KUKA KRL program: p01.src, p01.dat

--- p01.src ---
&ACCESS RV1
&REL 82
&COMMENT CX482 FHEV
&PARAM EDITMASK = *
&PARAM TEMPLATE = C:\KRC\Roboter\Template\vorgabe
&PARAM DISKPATH = KRC:\R1\Program\Main Programs
DEF p01( )
;================================================
;FOLD INI;%{PE}
  ;FOLD BASISTECH INI
    GLOBAL INTERRUPT DECL 3 WHEN $STOPMESS==TRUE DO IR_STOPM ( )
    INTERRUPT ON 3
    BAS (#INITMOV,0 )
  ;ENDFOLD (BASISTECH INI)
  ;FOLD USER INI
    ;Make your modifications here
BACKJUMP=FALSE
  ;ENDFOLD (USER INI)
;ENDFOLD (INI)
; MODEL     : CX482
; IE GROUP  : FHEV
; STATION   : ST105
; ROBOT     : 105R1
; FUNCTION  : GLUE ON FLANGE - 2C
;================================================

;Control TC
$TIMER[7]=0
$TIMER_STOP[7]=FALSE

;FOLD PTP HOME Vel=100 % DEFAULT;%{PE}%R 8.3.48,%MKUKATPBASIS,%CMOVE,%VPTP,%P 1:PTP, 2:HOME, 3:, 5:100, 7:DEFAULT
$BWDSTART=FALSE
PDAT_ACT=PDEFAULT
FDAT_ACT=FHOME
BAS(#PTP_PARAMS,100)
$H_POS=XHOME
PTP XHOME
;ENDFOLD

;FOLD Start Cycle Timer
$TIMER[1]=0
$TIMER_STOP[1]=FALSE
;ENDFOLD

INFOPOS:
;FOLD PTP P1wait Vel=100 % PDAT2 Tool[5] Base[0];%{PE}%R 8.3.48,%MKUKATPBASIS,%CMOVE,%VPTP,%P 1:PTP, 2:P1wait, 3:, 5:100, 7:PDAT2
$BWDSTART=FALSE
PDAT_ACT=PPDAT2
FDAT_ACT=FP1wait
BAS(#PTP_PARAMS,100)
PTP XP1wait
;ENDFOLD

;if false then

;FOLD TYPE INFO

O_TYPE_REQ=FALSE
WAIT FOR I_TYPE_INFO==0
O_TYPE_REQ=TRUE
WAIT FOR (I_TYPE_INFO>0)
O_TYPE_INFO=I_TYPE_INFO


;ENDFOLD

;rack1 o rack2

;endif

WAIT FOR ($IN[49]==TRUE) OR ($IN[50]==TRUE) OR ($IN[51]==TRUE)

cils_init()
IF $in[49]==TRUE THEN
   INDICE_RACK=1              ;Variable calculo TC
   P01pick1 ( )               ; PICK In Station XX
   IF I_Rethp THEN              ; Return To Home
     GOTO HOMEPOS
   ENDIF
   IF BACKJUMP THEN
     BACKJUMP=FALSE
     GOTO INFOPOS
   ENDIF
   IF CARTJUMP THEN              ; Return To Home
     GOTO HOMEPOS
   ENDIF

  ; P01drop()
   P01drop_new()

endif

IF $in[50]==TRUE THEN
   INDICE_RACK=2              ;Variable calculo TC
   P01pick2 ( )                ; PICK In Station XX
   IF I_Rethp THEN              ; Return To Home
     GOTO HOMEPOS
   ENDIF
   IF BACKJUMP THEN
     BACKJUMP=FALSE
     GOTO INFOPOS
   ENDIF
   IF CARTJUMP THEN              ; Return To Home
     GOTO HOMEPOS
   ENDIF
  ; P01drop()
   P01drop_new()

ENDIF


IF $in[51]==TRUE THEN

   P01pick3 ( )                ; PICK In carton XX


;FOLD OUT 21 'Area Release 5' State=TRUE ;%{PE}%R 8.3.48,%MKUKATPBASIS,%COUT,%VOUTX,%P 2:21, 3:Area Release 5, 5:TRUE, 6:
$OUT[21]=TRUE
;ENDFOLD
;FOLD TYPE INFO

O_TYPE_REQ=FALSE
WAIT FOR I_TYPE_INFO==0
O_TYPE_REQ=TRUE
WAIT FOR (I_TYPE_INFO>0)
POS_CARTON=I_TYPE_INFO
O_TYPE_INFO=I_TYPE_INFO
O_TYPE_REQ=FALSE

;ENDFOLD
   P01drop3 ( )                ; DROP In carton XX


   IF I_Rethp THEN              ; Return To Home
     GOTO HOMEPOS
   ENDIF
   IF BACKJUMP THEN
     BACKJUMP=FALSE
     GOTO INFOPOS
   ENDIF
   IF CARTJUMP THEN              ; Return To Home
     GOTO HOMEPOS
   ENDIF
  ; P01drop()
   ;P01drop_new()

ENDIF

If false then
; Solicitar fin de trabajo
;FOLD Fordtech.End_Work_Req ;%{PE}%MKUKATPUSER
END_WORK_REQ()
;ENDFOLD
endif

HOMEPOS:
;FOLD PTP HOME  Vel= 100 % DEFAULT;%{PE}%R 5.4.33,%MKUKATPBASIS,%CMOVE,%VPTP,%P 1:PTP, 2:HOME, 3:, 5:100, 7:DEFAULT
$BWDSTART=FALSE
PDAT_ACT=PDEFAULT
FDAT_ACT=FHOME
BAS(#PTP_PARAMS,100)
$H_POS=XHOME
PTP XHOME
;ENDFOLD

;FOLD Stop Cyclus Timer
$TIMER_STOP[1]=TRUE
$TIMER[6]=$TIMER[1]
;ENDFOLD

INIT_RS ( )                  ; Reset Job_Ready 1-8
INIT_EXT ( )                 ; Init Auto_Extern
END

--- p01.dat ---
&ACCESS RV1
&REL 82
&COMMENT CX482 FHEV
&PARAM EDITMASK = *
&PARAM TEMPLATE = C:\KRC\Roboter\Template\vorgabe
&PARAM DISKPATH = KRC:\R1\Program\Main Programs
DEFDAT  p01
;FOLD EXTERNAL DECLARATIONS;%{PE}%MKUKATPBASIS,%CEXT,%VCOMMON,%P
;FOLD GRIPPERTECH EXT
;EXT  H50 (INT  :IN,INT  :IN,INT  :IN,GRP_TYP  :IN )
;ENDFOLD (GRIPPERTECH EXT)
;FOLD SPOTTECH EXT
EXT  USERSPOT (S_COMMAND  :IN,SPOT_TYPE  :IN )
;ENDFOLD (SPOTTECH EXT)
;FOLD BASISTECH EXT;%{PE}%MKUKATPBASIS,%CEXT,%VEXT,%P
EXT  BAS (BAS_COMMAND  :IN,REAL  :IN )
DECL INT SUCCESS
;ENDFOLD (BASISTECH EXT)
;FOLD USER EXT;%{E}%MKUKATPUSER,%CEXT,%VEXT,%P
;Make your modifications here

;ENDFOLD (USER EXT)
;ENDFOLD (EXTERNAL DECLARATIONS)



DECL BASIS_SUGG_T LAST_BASIS={POINT1[] "P0                      ",POINT2[] "P0                      ",CP_PARAMS[] "CPDAT0                  ",PTP_PARAMS[] "PDAT0                   ",CONT[] "                        ",CP_VEL[] "2.0                     ",PTP_VEL[] " 100                    ",SYNC_PARAMS[] "SYNCDAT                 ",SPL_NAME[] "S0                      ",A_PARAMS[] "ADAT0                   "}
DECL E6AXIS XP01WAIR={A1 -25.4435329,A2 -130.127853,A3 135.595306,A4 3.03102922,A5 82.9436340,A6 -5.90488243,E1 0.0,E2 0.0,E3 0.0,E4 0.0,E5 0.0,E6 0.0}
DECL FDAT FP01WAIR={TOOL_NO 6,BASE_NO 1,IPO_FRAME #BASE,POINT2[] " ",TQ_STATE FALSE}
DECL PDAT PH={VEL 100.000,ACC 100.000,APO_DIST 100.000,APO_MODE #CDIS,GEAR_JERK 50.0000,EXAX_IGN 0}
DECL E6AXIS XP01WAIT={A1 -25.4435329,A2 -130.127853,A3 135.595306,A4 3.03102922,A5 82.9436340,A6 -5.90488243,E1 0.0,E2 0.0,E3 0.0,E4 0.0,E5 0.0,E6 0.0}
DECL FDAT FP01WAIT={TOOL_NO 6,BASE_NO 1,IPO_FRAME #BASE,POINT2[] " ",TQ_STATE FALSE}
DECL E6POS XP1wait={X 290.951233,Y 816.177124,Z 1275.55042,A -86.9976196,B 22.0779018,C -179.006119,S 6,T 27,E1 0.0,E2 0.0,E3 0.0,E4 0.0,E5 0.0,E6 0.0}
DECL FDAT FP1wait={TOOL_NO 5,BASE_NO 0,IPO_FRAME #BASE,POINT2[] " ",TQ_STATE FALSE}
DECL PDAT PPDAT1={VEL 100.000,ACC 100.000,APO_DIST 500.000,APO_MODE #CDIS,GEAR_JERK 100.000,EXAX_IGN 0}
DECL MODULEPARAM_T LAST_TP_PARAMS={PARAMS[] "Kuka.VelocityFieldEnabled=False; Kuka.ColDetectFieldEnabled=False; Kuka.MovementParameterFieldEnabled=False; Kuka.IsAngleEnabled=False; Kuka.PointName=P1wait; Kuka.FrameData.base_no=0; Kuka.FrameData.tool_no=1; Kuka.FrameData.ipo_frame=#BASE; Kuka.isglobalpoint=False; Kuka.MoveDataPtpName=PDAT1; Kuka.MovementDataPdat.apo_mode=#CDIS; Kuka.MovementDataPdat.apo_dist=500; Kuka.MovementData.vel=100; Kuka.MovementData.acc=100; Kuka.MovementData.exax_ign=0; Kuka.VelocityPtp=100; Kuka.BlendingEnabled=False; Kuka.APXEnabled=False; Kuka.CurrentCDSetIndex=0  "}
DECL PDAT PPDAT2={VEL 100.000,ACC 100.000,APO_DIST 100.000,GEAR_JERK 50.0000,EXAX_IGN 0}
ENDDAT
